Staubli VAL3: Socket1.dtx

public bool bCalibrating
public bool bTaskDetOK
num nLatchedValue
public num nMaxNumOfObject = 10
public num nNumOfPart = -1
num nObjectID = -1
sio skFromRobot
string sDetNum
string sErrorCode[6]
  [1] = "Could not convert to num ID"
  [2] = "Could not convert to num X"
  [3] = "Could not convert to num Y"
  [4] = "Could not convert to num RZ"
  [5] = "Could not convert to num Encoder Latched Value"
string sTASK
trsf trObjectPos
